Staubli VAL3: SaveData.pjx

--- SaveData.pjx ---
Parameters version=s7.8.3 stackSize=5000 millimeterUnit=true
Program file=start.pgx
Program file=stop.pgx
Data file=SaveData.dtx

--- SaveData.dtx ---
public bool bHome = true
public jointRx jJhome
public mdesc mNomSpeed
public num nPage_Traj = 1
public num nPage_editTraj = 7
public num nPage_viewTraj = 1
public pointRx pPoinTest[8]
  [0] = {x=32, y=32, fatherId=world[0]}
  [1] = {x=44, y=98, z=99, rx=55, ry=33, rz=22, fatherId=world[0]}
  [2] = {x=332, y=23, z=2, rx=23, ry=22, fatherId=world[0]}
  [3] = {y=34, rx=23, fatherId=world[0]}
  [4] = {x=12, y=22, z=90, rx=23, ry=23, rz=23, fatherId=world[0]}
  [5] = {x=11, z=44, rx=34, ry=12, rz=23, fatherId=world[0]}
  [6] = {x=2, y=22, z=4, rx=2, ry=33, rz=11, fatherId=world[0]}
  [7] = {x=23, fatherId=world[0]}
public string sTest

--- changeSession.pgx ---
public program changeSession(string x_sName)
  local string l_sPathTraj
  local string l_sPathProg
  local string l_sRootPath
  local string l_sPathCycle
  local string l_sPathSave
  local num i
begin
  //
  // change the session
  //
  // check if the robot is empty
  if (isEmpty()and isSettled())and watch(bToReload==false,120)==true
    if x_sName!="template"
      l_sPathTraj="saveTraj/"
      l_sPathProg="saveProg/"
      l_sPathSave="saveCycle/"
      l_sRootPath="Disk://session/"+x_sName+"/"
      // trajectory
      sPathTraj=l_sRootPath+l_sPathTraj
      // program
      sPathProg=l_sRootPath+l_sPathProg
      // process list
      sPathPList=l_sRootPath+l_sPathSave
      // save it
      sSession=x_sName
    else
      // trajectory
      sPathTraj="kernel/template/session/saveTraj/"
      // program
      sPathProg="kernel/template/session/saveProg/"
      // process list
      sPathPList="kernel/template/session/saveCycle/"
    endIf
    // reaload all...
    bToReload=true
    // watch it
    if watch(bToReload==false,120)==false
      popUpMsg("ERROR TIMEOUT!!! LOADING SESSION ...")
      logMsg("ERROR LOADING SESSION ...")
      wait(bToReload==false)
    endIf
  else
    popUpMsg("Error while changing the session the robot is working...")
    logMsg("Error while changing the session the robot is working...")
    delay(1)
  endIf
end

--- getListSession.pgx ---
public program getListSession(string& x_sSession[] (dimensions=1))
begin
  // Build the list
  libList("session",x_sSession)
end

--- getPathInstr.pgx ---
public program getPathInstr(string x_sInstr (dimensions=1), string& x_sPath (dimensions=1))
begin
  // give back the path of the Instruction
  if isDefined(iInstruction[x_sInstr])
    x_sPath=iInstruction[x_sInstr].sPath
  else
    x_sPath=""
  endIf
end

--- getSession.pgx ---
public program getSession(string& x_sName[] (dimensions=1))
  local num l_nPos[2]
  local num l_nSize
begin
  l_nPos=find(sPathTraj,"Disk://session")
  if l_nPos==-1
    // give back the session name
    x_sName=""
  else
    l_nPos[1]=find(sPathTraj,"/saveTraj/")
    l_nSize=l_nPos[1]-l_nPos-len("Disk://session/")
    x_sName=mid(sPathTraj,l_nSize,l_nPos+len("Disk://session/"))
  endIf
end

--- getTool.pgx ---
public program getTool(tool& x_tTool[] (dimensions=1), num x_nIndex (dimensions=1))
begin
  // get the tool
  x_tTool=tData[x_nIndex].tcp
end
